TYPE stServo :
STRUCT
	x : REAL;
	y : REAL;
	radius : REAL;
END_STRUCT
END_TYPE

(* stored: Version 1.1.0.1, ProductVersion 3.1.4026.8
   DUT stServo: Id {f177b22d-5767-48cd-a3a5-5275a012b774} *)
